ADAPTER SubscribeEventAdp (* Subscribe event adapter *)
  (* Standard: 61499-2; Description: Copyright (c) 2019 fortiss GmbH This program and the accompanying materials are made available under the terms of the Eclipse Public License 2.0 which is available at https://www.eclipse.org/legal/epl-2.0/ SPDX-License-Identifier: EPL-2.0 *)
  (* Version 1.0, 2019-09-18, Cabral, fortiss GmbH *)
  (* Compiler header: package fb.test; *)
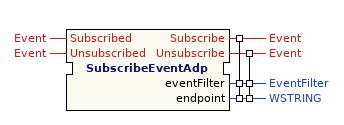
  EVENT_INPUT
    Subscribed; (* Subscribe finished *)
    Unsubscribed; (* Unsubscribe finished *)
  END_EVENT
  EVENT_OUTPUT
    Subscribe WITH eventFilter, endpoint; (* Subscribe to event *)
    Unsubscribe WITH endpoint, eventFilter; (* Unsubscribe from event *)
  END_EVENT
  VAR_OUTPUT
    eventFilter : EventFilter; (* Event filter *)
    endpoint : WSTRING; (* Endpoint (IP:PORT/URI) of the Service Registry (not officially in the documentation, but it simplifies the FBs) *)
  END_VAR
  SERVICE SOCKET/PLUG (* Subscribe event adapter *)
    SEQUENCE request_confirm
      SOCKET.REQ(REQD) -> PLUG.REQ(REQD);
      PLUG.CNF(CNFD) -> SOCKET.CNF(CNFD);
    END_SEQUENCE
    SEQUENCE indication_response
      PLUG.IND(INDD) -> SOCKET.IND(INDD);
      SOCKET.RSP(RSPD) -> PLUG.RSP(RSPD);
    END_SEQUENCE
  END_SERVICE
END_ADAPTER
